FUNCTION_BLOCK _ETcVnBorderInterpolationMethod_TestSuite EXTENDS TcUnit.FB_TestSuite
VAR
END_VAR

TestAddress();
TestClearReference();
TestClone();
TestTypeNameReturnsExpected();
TestIdentifierReturnsExpected();
TestMakeReferenceToFollowsReference();
TestMakeReferenceToUpdatesReference();
TestSize();
TestValueReturnsExpectedAfterInit();
TestValueReturnsExpectedAfterChange();
TestSerializeTypeWith();
TestSerializeWith();
TestTryDeserializeFrom();
TestTryMakeReferenceToFollowsReference();
TestTryMakeReferenceToUpdatesReference();

METHOD PUBLIC TestAddress
VAR
    _type : _ETcVnBorderInterpolationMethod(ETcVnBorderInterpolationMethod.TCVN_BIM_CONSTANT);
    notExpected : PVOID := 0;
    actual : PVOID;
END_VAR
TEST('TestAddress');

actual := _type.Address;

AssertFalse(
    Condition := (notExpected = actual),
    Message := 'Type did not return a valid address.'
);

TEST_FINISHED();
END_METHOD

METHOD PUBLIC TestClearReference
VAR
    _type : _ETcVnBorderInterpolationMethod(ETcVnBorderInterpolationMethod.TCVN_BIM_CONSTANT);
	target : ETcVnBorderInterpolationMethod := ETcVnBorderInterpolationMethod.TCVN_BIM_CONSTANT;
    expected : ETcVnBorderInterpolationMethod := ETcVnBorderInterpolationMethod.TCVN_BIM_CONSTANT;
    actual : ETcVnBorderInterpolationMethod;
END_VAR
TEST('TestClearReference');

_type.MakeReferenceTo(target);
_type.ClearReference();
target := ETcVnBorderInterpolationMethod.TCVN_BIM_REPLICATE;

actual := _type.Value;

AssertEquals(
    Expected := expected,
    Actual := actual,
    Message := 'Value continued to follow target.'
);

TEST_FINISHED();
END_METHOD

METHOD PUBLIC TestClone
VAR
    _type : _ETcVnBorderInterpolationMethod(ETcVnBorderInterpolationMethod.TCVN_BIM_CONSTANT);
	clone : I_Datatype;
	isValidClone : BOOL;
	compareResult : DINT;
END_VAR
TEST('TestClone');

clone := _type.Clone();

isValidClone := clone <> 0;

IF isValidClone THEN
	compareResult := memcmp(_type.Address, clone.Address, clone.Size);
END_IF

AssertTrue(
	Condition := isValidClone,
	Message := 'Clone did not produce a clone'
);

AssertEquals_DINT(
	Expected := 0,
    Actual := compareResult,
    Message := 'Clone did not return a valid clone.'
);

clone.Dispose();

TEST_FINISHED();
END_METHOD

METHOD PUBLIC TestIdentifierReturnsExpected
VAR
    _type : _ETcVnBorderInterpolationMethod(ETcVnBorderInterpolationMethod.TCVN_BIM_CONSTANT);
    expected : STRING := 'ETcVnBorderInterpolationMethod';
    actual : STRING;
END_VAR
TEST('TestIdentifierReturnsExpected');

actual := _type.Identifier;

AssertEquals_STRING(
    Expected := expected,
    Actual := actual,
    Message := 'Type did not return correct iec type.'
);

TEST_FINISHED();
END_METHOD

METHOD PUBLIC TestMakeReferenceToFollowsReference
VAR
    _type : _ETcVnBorderInterpolationMethod(ETcVnBorderInterpolationMethod.TCVN_BIM_CONSTANT);
	target : ETcVnBorderInterpolationMethod := ETcVnBorderInterpolationMethod.TCVN_BIM_CONSTANT;
    expected : ETcVnBorderInterpolationMethod := ETcVnBorderInterpolationMethod.TCVN_BIM_REPLICATE;
    actual : ETcVnBorderInterpolationMethod;
END_VAR
TEST('TestMakeReferenceToFollowsReference');

_type.MakeReferenceTo(target);
target := ETcVnBorderInterpolationMethod.TCVN_BIM_REPLICATE;

actual := _type.Value;

AssertEquals(
    Expected := expected,
    Actual := actual,
    Message := 'Value did not follow target change.'
);

TEST_FINISHED();
END_METHOD

METHOD PUBLIC TestMakeReferenceToUpdatesReference
VAR
    _type : _ETcVnBorderInterpolationMethod(ETcVnBorderInterpolationMethod.TCVN_BIM_CONSTANT);
	target : ETcVnBorderInterpolationMethod := ETcVnBorderInterpolationMethod.TCVN_BIM_CONSTANT;
    expected : ETcVnBorderInterpolationMethod := ETcVnBorderInterpolationMethod.TCVN_BIM_REPLICATE;
    actual : ETcVnBorderInterpolationMethod;
END_VAR
TEST('TestMakeReferenceToUpdatesReference');

_type.MakeReferenceTo(target);
_type.Value := ETcVnBorderInterpolationMethod.TCVN_BIM_REPLICATE;

actual := target;

AssertEquals(
    Expected := expected,
    Actual := actual,
    Message := 'Value did not update target.'
);

TEST_FINISHED();
END_METHOD

METHOD PUBLIC TestSerializeTypeWith
VAR
    _type : _ETcVnBorderInterpolationMethod(ETcVnBorderInterpolationMethod.TCVN_BIM_CONSTANT);
    serializer : JsonSerializer;
    expected : STRING(500) := '{"typeName":"ENUM","identifier":"ETcVnBorderInterpolationMethod","enumerations":["TCVN_BIM_CONSTANT","TCVN_BIM_REPLICATE","TCVN_BIM_REFLECT","TCVN_BIM_WRAP","TCVN_BIM_REFLECT_101","TCVN_BIM_DEFAULT","TCVN_BIM_TRANSPARENT","TCVN_BIM_ISOLATED_CONSTANT","TCVN_BIM_ISOLATED_REPLICATE","TCVN_BIM_ISOLATED_REFLECT","TCVN_BIM_ISOLATED_WRAP","TCVN_BIM_ISOLATED_REFLECT_101"],"baseType":{"typeName":"DINT","minValue":-2147483648,"maxValue":2147483647,"isSigned":true,"isFloat":false}}'; 
    actual : STRING(500);
END_VAR
TEST('TestSerializeTypeWith');

serializer.Reset();
_type.SerializeTypeWith(serializer);
serializer.TryGetSerializedData(ADR(actual), SIZEOF(actual));

AssertEquals_STRING(
    Expected := expected,
    Actual := actual,
    Message := 'Serialization of type did not return correct string.'
);

TEST_FINISHED();
END_METHOD

METHOD PUBLIC TestSerializeWith
VAR
    _type : _ETcVnBorderInterpolationMethod(ETcVnBorderInterpolationMethod.TCVN_BIM_CONSTANT);
    serializer : JsonSerializer;
    expected : STRING := '"TCVN_BIM_CONSTANT"';
    actual : STRING(500);
END_VAR
TEST('TestSerializeWith');

serializer.Reset();
_type.SerializeWith(serializer);
serializer.TryGetSerializedData(ADR(actual), SIZEOF(actual));

AssertEquals_STRING(
    Expected := expected,
    Actual := actual,
    Message := 'Serialization of type data did not return correct string.'
);

TEST_FINISHED();
END_METHOD

METHOD PUBLIC TestSize
VAR
    _type : _ETcVnBorderInterpolationMethod(ETcVnBorderInterpolationMethod.TCVN_BIM_CONSTANT);
    expected : UDINT := SIZEOF(ETcVnBorderInterpolationMethod);
    actual : UDINT;
END_VAR
TEST('TestSize');

actual := _type.Size;

AssertEquals_UDINT(
    Expected := Expected,
    Actual := actual,
    Message := 'Type did not return the correct size.'
);

TEST_FINISHED();
END_METHOD

METHOD PUBLIC TestTryDeserializeFrom
VAR
    deserializer : JsonDeserializer;
    feedback : DeserializerFeedback;
    json : STRING := '"TCVN_BIM_CONSTANT"';
    _type : _ETcVnBorderInterpolationMethod(ETcVnBorderInterpolationMethod.TCVN_BIM_CONSTANT);
    expected : ETcVnBorderInterpolationMethod := ETcVnBorderInterpolationMethod.TCVN_BIM_CONSTANT;
    actual : ETcVnBorderInterpolationMethod;
 END_VAR
TEST('TestTryDeserializeFrom');

deserializer.Reset();
deserializer.TryLoad(json);
_type.TryDeserializeFrom(Deserializer, Feedback);

actual := _type.Value;

AssertEquals(
    Expected := expected,
    Actual := actual,
    Message := 'Type did not deserialize correctly.'
);

TEST_FINISHED();
END_METHOD

METHOD PUBLIC TestTryMakeReferenceToFollowsReference
VAR
    _type : _ETcVnBorderInterpolationMethod(ETcVnBorderInterpolationMethod.TCVN_BIM_CONSTANT);
	target : _ETcVnBorderInterpolationMethod(ETcVnBorderInterpolationMethod.TCVN_BIM_CONSTANT);
    expected : ETcVnBorderInterpolationMethod := ETcVnBorderInterpolationMethod.TCVN_BIM_REPLICATE;
    actual : ETcVnBorderInterpolationMethod;
END_VAR
TEST('TestTryMakeReferenceToFollowsReference');

_type.TryMakeReferenceTo(target);
target.Value := ETcVnBorderInterpolationMethod.TCVN_BIM_REPLICATE;

actual := _type.Value;

AssertEquals(
    Expected := expected,
    Actual := actual,
    Message := 'Value did not follow target change.'
);

TEST_FINISHED();
END_METHOD

METHOD PUBLIC TestTryMakeReferenceToUpdatesReference
VAR
    _type : _ETcVnBorderInterpolationMethod(ETcVnBorderInterpolationMethod.TCVN_BIM_CONSTANT);
	target : _ETcVnBorderInterpolationMethod(ETcVnBorderInterpolationMethod.TCVN_BIM_CONSTANT);
    expected : ETcVnBorderInterpolationMethod := ETcVnBorderInterpolationMethod.TCVN_BIM_REPLICATE;
    actual : ETcVnBorderInterpolationMethod;
END_VAR
TEST('TestTryMakeReferenceToUpdatesReference');

_type.TryMakeReferenceTo(target);
_type.Value := ETcVnBorderInterpolationMethod.TCVN_BIM_REPLICATE;

actual := target.Value;

AssertEquals(
    Expected := expected,
    Actual := actual,
    Message := 'Value did not update target.'
);

TEST_FINISHED();
END_METHOD

METHOD PUBLIC TestTypeNameReturnsExpected
VAR
    _type : _ETcVnBorderInterpolationMethod(ETcVnBorderInterpolationMethod.TCVN_BIM_CONSTANT);
    expected : STRING := 'ENUM';
    actual : STRING;
END_VAR
TEST('TestTypeNameReturnsExpected');

actual := _type.TypeName;

AssertEquals_STRING(
    Expected := expected,
    Actual := actual,
    Message := 'Type did not return correct iec type.'
);

TEST_FINISHED();
END_METHOD

METHOD PUBLIC TestValueReturnsExpectedAfterChange
VAR
    _type : _ETcVnBorderInterpolationMethod(ETcVnBorderInterpolationMethod.TCVN_BIM_CONSTANT);
    expected : ETcVnBorderInterpolationMethod := ETcVnBorderInterpolationMethod.TCVN_BIM_REPLICATE;
    actual : ETcVnBorderInterpolationMethod;
END_VAR
TEST('TestValueReturnsExpectedAfterChange');

_type.Value := ETcVnBorderInterpolationMethod.TCVN_BIM_REPLICATE;

actual := _type.Value;

AssertEquals(
    Expected := expected,
    Actual := actual,
    Message := 'Expected value not returned after change.'
);

TEST_FINISHED();
END_METHOD

METHOD PUBLIC TestValueReturnsExpectedAfterInit
VAR
    _type : _ETcVnBorderInterpolationMethod(ETcVnBorderInterpolationMethod.TCVN_BIM_CONSTANT);
    expected : ETcVnBorderInterpolationMethod := ETcVnBorderInterpolationMethod.TCVN_BIM_CONSTANT;
    actual : ETcVnBorderInterpolationMethod;
END_VAR
TEST('TestValueReturnsExpectedAfterInit');

actual := _type.Value;

AssertEquals(
    Expected := expected,
    Actual := actual,
    Message := 'Expected value not returned after Init.'
);

TEST_FINISHED();
END_METHOD

END_FUNCTION_BLOCK

(* stored: Version 1.1.0.1, ProductVersion 3.1.4024.12
   POU _ETcVnBorderInterpolationMethod_TestSuite: Id {0611783b-ff20-0cc7-004a-e1e7a5e20d24}, SpecialFunc None
   Method TestAddress: Id {5b3262e4-be8d-0932-103f-9d27cfff273d}
   Method TestClearReference: Id {fa206519-2e05-06aa-11cf-65766ccef94c}
   Method TestClone: Id {a475de12-2057-05f4-1964-fd1fbee156fe}
   Method TestIdentifierReturnsExpected: Id {67d0c7c2-dc69-0abd-10a9-125670161568}
   Method TestMakeReferenceToFollowsReference: Id {f4d289a9-20bb-0a97-0d63-025395aa1367}
   Method TestMakeReferenceToUpdatesReference: Id {5f38e24b-8504-0dcf-1590-971ed4671812}
   Method TestSerializeTypeWith: Id {f91980b8-d533-0539-1c6a-c682e75f9a86}
   Method TestSerializeWith: Id {5062eb24-9862-07a2-155f-7a4b73620699}
   Method TestSize: Id {9b10773a-286f-0acd-1eb0-0dd397cfbf6b}
   Method TestTryDeserializeFrom: Id {1569a90e-35f1-0a2a-1e91-a59e38f61be1}
   Method TestTryMakeReferenceToFollowsReference: Id {a6cf6316-76bd-006e-14f1-c319e8bd023b}
   Method TestTryMakeReferenceToUpdatesReference: Id {f1d53e55-25da-0d92-012d-31dabed5f843}
   Method TestTypeNameReturnsExpected: Id {a49b2e91-652c-0fc6-2012-3d0abb1d85e8}
   Method TestValueReturnsExpectedAfterChange: Id {49343caf-75e6-0e50-118b-ae53b5cf1832}
   Method TestValueReturnsExpectedAfterInit: Id {fd235e20-16ae-04f8-3d1d-70e98a9c28b0} *)
